// TIA Portal V20 export
VAR_GLOBAL   // PLC tag table "LKinCtrl_HMI_Shared_OperationModes"
END_VAR
VAR_GLOBAL CONSTANT   // user constants
   LKINCTRL_OPERATION_MODE_MANUAL : Int := 2;   // Operation mode "Manual".
   LKINCTRL_OPERATION_MODE_AUTO : Int := 1;   // Operation mode "Automatic".
   LKINCTRL_OPERATION_MODE_NOP : Int := 10;   // Operation mode "No operation". HMI is locked.
   LKINCTRL_OPERATION_MODE_TEST_RUN : Int := 3;   // Operation mode "Test run".
   LKINCTRL_OPERATION_MODE_FULL_OPERATION : Int := 0;   // Operation mode "Full operation". No restriction in HMI.
END_VAR
